{attribute 'GeneratedUsingTerminal: EL3041-0000-0017'}
{attribute addProperty BoxType "EL3041-0000-0017"}
{attribute addProperty Description "EL3041 1Ch. Ana. Input 0-20mA"}
{attribute addProperty Physics "KK"}
{attribute addProperty Id "AI_StandardAT %I*AI_Standard_Channel_4A3944819WcStateAT %I*WcState_9091E0EB2InfoDataAT %I*InfoData_32EB74EA10"}
{attribute addProperty CRC "3794663976"}
{attribute addProperty Size "21"}
TYPE EL3041_E22DFA28 EXTENDS EtcSlaveTerminalBase_947E5A46 :
STRUCT
	{attribute addProperty Name "AI_Standard"}
	AI_Standard : AI_Standard_Channel_4A394481;
	{attribute addProperty Name "WcState"}
	WcState : WcState_9091E0EB;
	{attribute addProperty Name "InfoData"}
	InfoData : InfoData_32EB74EA;
END_STRUCT
END_TYPE

(* stored: Version 1.2.0.0, ProductVersion 3.1.4024.9
   DUT EL3041_E22DFA28: Id {f4d03a86-fa01-436f-b86c-ecb9d7edf8aa} *)
